// TIA Portal project "Project1" (V18)
// memory addressing

(* hardware
DEVICE "S7-1200 station_1"  S7-1200 Station
   slot 0: "Rack_0"  S7-1200 Rack  Rack  V1.0
   slot 1: "PLC_1"  CPU 1211C DC/DC/DC  6ES7 211-1AE40-0XB0  V4.6
*)

// ===== PLC "PLC_1"  CPU 1211C DC/DC/DC =====

VAR_GLOBAL   // PLC tag table "Default tag table"
   "CW" AT %I0.0 : Bool;
   "CCW" AT %I0.1 : Bool;
   "MOTOR_R_CW" AT %Q0.0 : Bool;
   "STOP" AT %I0.2 : Bool;
   "Tag_1" AT %M0.0 : Bool;
   "MOTOR_R_CCW" AT %Q0.1 : Bool;
   "Tag_2" AT %M0.1 : Bool;
   "Tag_3" AT %M0.2 : Bool;
   "Tag_4" AT %M0.3 : Bool;
END_VAR

// folder: System blocks/Program resources

DATA_BLOCK "IEC_Timer_0_DB"   // DB1
{ S7_Optimized_Access := 'TRUE' }
AUTHOR : Simatic
FAMILY : IEC
NAME : IEC_TMR
VERSION : 1.0
// stored: InstanceOfName IEC_TIMER
"IEC_TIMER"
BEGIN
END_DATA_BLOCK

// folder: (top level)

ORGANIZATION_BLOCK "Main"   // OB1, LAD, ProgramCycle
TITLE = "Main Program Sweep (Cycle)"
{ S7_Optimized_Access := 'TRUE' }
VERSION : 0.1
// Tank_0_Level_Controller
   VAR_INPUT
      Initial_Call : Bool;   // Initial call of this OB
      Remanence : Bool;   // =True, if remanent data are available
   END_VAR
BEGIN

REGION Network 1
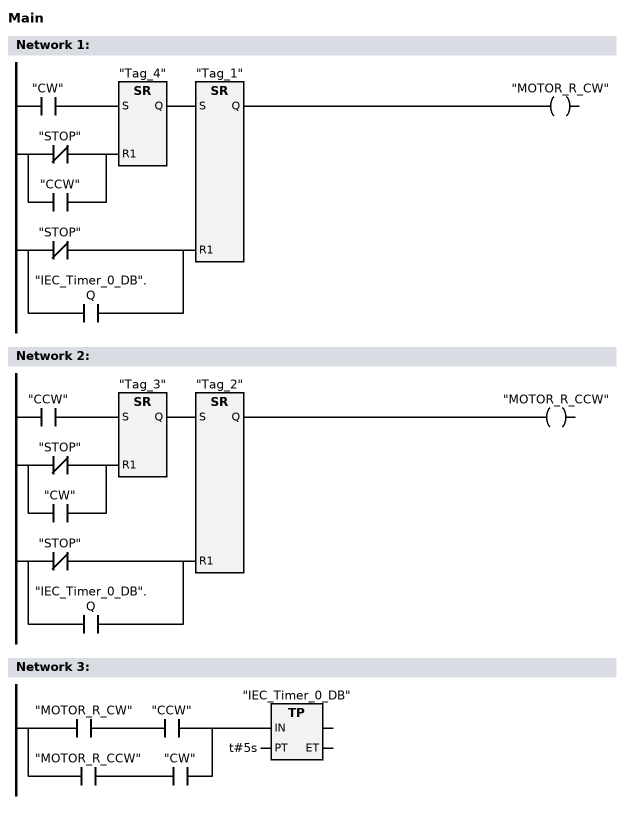
   RUNG wire#powerrail
      Contact( "CW" )
      S_SR(operand := "Tag_4", r1 := wire#w1)
      S_SR(operand := "Tag_1", r1 := wire#w2)
      Coil( "MOTOR_R_CW" )
   END_RUNG
   RUNG wire#powerrail
      I_Contact( "STOP" )
   END_RUNG wire#w1
   RUNG wire#powerrail
      Contact( "CCW" )
   END_RUNG wire#w1
   RUNG wire#powerrail
      I_Contact( "STOP" )
   END_RUNG wire#w2
   RUNG wire#powerrail
      Contact( "IEC_Timer_0_DB".Q )
   END_RUNG wire#w2
   // the same network as SCL:
   IF "CW" THEN
       "Tag_4" := TRUE;   // SR flip-flop
   END_IF;
   IF NOT "STOP" OR "CCW" THEN "Tag_4" := FALSE; END_IF;
   IF "Tag_4" THEN
       "Tag_1" := TRUE;   // SR flip-flop
   END_IF;
   IF NOT "STOP" OR "IEC_Timer_0_DB".Q THEN "Tag_1" := FALSE; END_IF;
   "MOTOR_R_CW" := "Tag_1";
END_REGION

REGION Network 2
   RUNG wire#powerrail
      Contact( "CCW" )
      S_SR(operand := "Tag_3", r1 := wire#w1)
      S_SR(operand := "Tag_2", r1 := wire#w2)
      Coil( "MOTOR_R_CCW" )
   END_RUNG
   RUNG wire#powerrail
      I_Contact( "STOP" )
   END_RUNG wire#w1
   RUNG wire#powerrail
      Contact( "CW" )
   END_RUNG wire#w1
   RUNG wire#powerrail
      I_Contact( "STOP" )
   END_RUNG wire#w2
   RUNG wire#powerrail
      Contact( "IEC_Timer_0_DB".Q )
   END_RUNG wire#w2
   // the same network as SCL:
   IF "CCW" THEN
       "Tag_3" := TRUE;   // SR flip-flop
   END_IF;
   IF NOT "STOP" OR "CW" THEN "Tag_3" := FALSE; END_IF;
   IF "Tag_3" THEN
       "Tag_2" := TRUE;   // SR flip-flop
   END_IF;
   IF NOT "STOP" OR "IEC_Timer_0_DB".Q THEN "Tag_2" := FALSE; END_IF;
   "MOTOR_R_CCW" := "Tag_2";
END_REGION

REGION Network 3
   "IEC_Timer_0_DB".TP(IN := ("MOTOR_R_CW" AND "CCW") OR ("MOTOR_R_CCW" AND "CW"), PT := t#5s);
END_REGION
END_ORGANIZATION_BLOCK